{attribute 'qualified_only'}
{attribute 'strict'}
TYPE Modes :
(
	STOP_EM := 0,
	STOP_OP := 1,
	AUTO := 2,
	MAN := 3,
	Stopping := 4
);
END_TYPE

(* stored: Version 1.1.0.1, ProductVersion 3.1.4024.9
   DUT Modes: Id {4c120f58-514b-4706-9a13-17782296efc4} *)
